{attribute addProperty BoxType "EK1100-0000-0018"}
{attribute addProperty Id "Beckhoff_EL1xxxEK1122Beckhoff_EL1xxxEK1122_BA3F35BD162A_0001_EL1002_0000_0000EL1002_FE5AE676486A_0002_EL1002_0000_0016EL1002_FE5AE676486A_0003_EL1002_0000_0017EL1002_FE5AE676486A_0004_EL1002_0000_0018EL1002_FE5AE676486A_0005_EL1004_0000_0000EL1004_5A15FBDA648A_0006_EL1004_0000_0016EL1004_5A15FBDA648A_0007_EL1004_0000_0017EL1004_5A15FBDA648A_0008_EL1004_0000_0018EL1004_5A15FBDA648A_0009_EL1004_0000_0019EL1004_5A15FBDA648A_0010_EL1004_0010_0000EL1004_5A15FBDA648A_0011_EL1004_0010_0016EL1004_5A15FBDA648A_0012_EL1004_0010_0017EL1004_5A15FBDA648A_0013_EL1004_0010_0018EL1004_5A15FBDA648A_0014_EL1004_0020_0016EL1004_5A15FBDA648A_0015_EL1008_0000_0016EL1008_C6161DDF9612A_0016_EL1008_0000_0017EL1008_C6161DDF9612A_0017_EL1008_0000_0018EL1008_C6161DDF9612A_0018_EL1012_0000_0000EL1012_FE5AE676486A_0019_EL1012_0000_0016EL1012_FE5AE676486A_0020_EL1012_0000_0017EL1012_FE5AE676486A_0021_EL1012_0000_0018EL1012_FE5AE676486A_0022_EL1014_0000_0000EL1014_5A15FBDA648A_0023_EL1014_0000_0016EL1014_5A15FBDA648A_0024_EL1014_0000_0017EL1014_5A15FBDA648A_0025_EL1014_0000_0018EL1014_5A15FBDA648A_0026_EL1014_0000_0019EL1014_5A15FBDA648A_0027_EL1014_0010_0000EL1014_5A15FBDA648A_0028_EL1014_0010_0016EL1014_5A15FBDA648A_0029_EL1014_0010_0017EL1014_5A15FBDA648A_0030_EL1014_0010_0018EL1014_5A15FBDA648A_0031_EL1014_0010_0019EL1014_5A15FBDA648A_0032_EL1018_0000_0016EL1018_C6161DDF9612A_0033_EL1018_0000_0017EL1018_C6161DDF9612A_0034_EL1018_0000_0018EL1018_C6161DDF9612A_0035_EL1024_0000_0016EL1024_5A15FBDA648A_0036_EL1024_0000_0017EL1024_5A15FBDA648A_0037_EL1024_0000_0018EL1024_5A15FBDA648A_0038_EL1034_0000_0016EL1034_5A15FBDA648A_0039_EL1034_0000_0017EL1034_5A15FBDA648A_0040_EL1034_0000_0018EL1034_5A15FBDA648A_0041_EL1052_0000_0016EL1052_0A1DBF07648A_0042_EL1054_0000_0016EL1054_0581C7AF9612A_0043_EL1084_0000_0016EL1084_5A15FBDA648A_0044_EL1084_0000_0017EL1084_5A15FBDA648A_0045_EL1084_0000_0018EL1084_5A15FBDA648A_0046_EL1088_0000_0016EL1088_C6161DDF9612A_0047_EL1088_0000_0017EL1088_C6161DDF9612A_0048_EL1088_0000_0018EL1088_C6161DDF9612A_0049_EL1094_0000_0016EL1094_5A15FBDA648A_0050_EL1094_0000_0017EL1094_5A15FBDA648A_0051_EL1094_0000_0018EL1094_5A15FBDA648A_0052_EL1098_0000_0016EL1098_C6161DDF9612A_0053_EL1098_0000_0017EL1098_C6161DDF9612A_0054_EL1098_0000_0018EL1098_C6161DDF9612A_0055_EL1104_0000_0016EL1104_5A15FBDA648A_0056_EL1104_0000_0017EL1104_5A15FBDA648A_0057_EL1104_0000_0018EL1104_5A15FBDA648A_0058_EL1114_0000_0016EL1114_5A15FBDA648A_0059_EL1114_0000_0017EL1114_5A15FBDA648A_0060_EL1114_0000_0018EL1114_5A15FBDA648A_0061_EL1124_0000_0016EL1124_5A15FBDA648A_0062_EL1124_0000_0017EL1124_5A15FBDA648A_0063_EL1124_0000_0018EL1124_5A15FBDA648A_0064_EL1134_0000_0016EL1134_5A15FBDA648A_0065_EL1134_0000_0017EL1134_5A15FBDA648A_0066_EL1134_0000_0018EL1134_5A15FBDA648A_0067_EL1144_0000_0016EL1144_5A15FBDA648A_0068_EL1144_0000_0017EL1144_5A15FBDA648A_0069_EL1144_0000_0018EL1144_5A15FBDA648A_0070_EL1202_0000_0016EL1202_FE5AE676486A_0071_EL1202_0000_0017EL1202_FE5AE676486A_0072_EL1202_0000_0018EL1202_FE5AE676486A_0073_EL1202_0000_0019EL1202_FE5AE676486A_0074_EL1202_0100_0016EL1202_3E03878817622A_0075_EL1202_0100_0017EL1202_3E03878817622A_0076_EL1202_0100_0018EL1202_3E03878817622A_0077_EL1202_0100_0019EL1202_3E03878817622A_0078_EL1252_0000_0017EL1252_30076DEE38448A_0079_EL1252_0000_0018EL1252_54261E5238448A_0080_EL1252_0000_0019EL1252_54261E5238448A_0081_EL1252_0000_0020EL1252_54261E5238448A_0082_EL1252_0000_0021EL1252_54261E5238448A_0083_EL1252_0000_0022EL1252_54261E5238448A_0084_EL1252_0010_0019EL1252_54261E5238448A_0085_EL1252_0010_0020EL1252_54261E5238448A_0086_EL1252_0010_0021EL1252_54261E5238448A_0087_EL1252_0050_0016EL1252_54261E5238448A_0088_EL1252_0050_0017EL1252_54261E5238448A_0089_EL1252_0050_0018EL1252_54261E5238448A_0090_EL1254_0000_0000EL1254_D71D85A467284A_0091_EL1262_0000_0002EL1262_0572C52632040A_0092_EL1262_0000_0003EL1262_0572C52632040A_0093_EL1262_0050_0002EL1262_0572C52632040A_0094_EL1262_0050_0003EL1262_0572C52632040A_0095_EL1258_0000_0016EL1258_54C5F1D75784723A_0096_EL1258_0000_0017EL1258_D5DBF8D73488436A_0097_EL1258_0010_0017EL1258_F90AE7941184148A_0098_EL1259_0000_0016EL1259_07379E76112401405A_0099_EL1259_0000_0017EL1259_CA442E63111841398A_0100_EL1259_0000_0018EL1259_0CA51D3C101201265A_0101_EL1382_0000_0016EL1382_0A1DBF07648A_0102_EL1382_0000_0017EL1382_0A1DBF07648A_0103_EL1382_0000_0018EL1382_0A1DBF07648A_0104_EL1702_0000_0016EL1702_FE5AE676486A_0105_EL1702_0000_0017EL1702_FE5AE676486A_0106_EL1702_0020_0016EL1702_FE5AE676486A_0107_EL1712_0000_0016EL1712_FE5AE676486A_0108_EL1712_0020_0016EL1712_FE5AE676486A_0109_EL1722_0000_0016EL1722_FE5AE676486A_0110_EL1722_0000_0017EL1722_FE5AE676486A_0111_EL1804_0000_0016EL1804_5A15FBDA648A_0112_EL1804_0000_0017EL1804_5A15FBDA648A_0113_EL1804_0000_0018EL1804_5A15FBDA648A_0114_EL1808_0000_0016EL1808_C6161DDF9612A_0115_EL1808_0000_0017EL1808_C6161DDF9612A_0116_EL1808_0000_0018EL1808_C6161DDF9612A_0117_EL1809_0000_0016EL1809_8059E62316020A_0118_EL1809_0000_0017EL1809_8059E62316020A_0119_EL1809_0000_0018EL1809_8059E62316020A_0120_EL1814_0000_0016EL1814_5A15FBDA648A_0121_EL1814_0000_0017EL1814_5A15FBDA648A_0122_EL1814_0000_0018EL1814_5A15FBDA648A_0123_EL1819_0000_0016EL1819_8059E62316020A_0124_EL1819_0000_0017EL1819_8059E62316020A_0125_EL1819_0000_0018EL1819_8059E62316020A_0126_EL1852_0000_0016EL1852_6598BC3916020A_0127_EL1859_0000_0016EL1859_6598BC3916020A_0128_EL1859_0000_0017EL1859_6598BC3916020A_0129_EL1859_0000_0018EL1859_6598BC3916020A_0130_EL1862_0000_0016EL1862_8059E62316020A_0131_EL1862_0000_0017EL1862_8059E62316020A_0132_EL1862_0000_0018EL1862_8059E62316020A_0133_EL1862_0000_0019EL1862_8059E62316020A_0134_EL1862_0010_0016EL1862_8059E62316020A_0135_EL1862_0010_0017EL1862_8059E62316020A_0136_EL1862_0010_0018EL1862_8059E62316020A_0137_EL1862_0010_0019EL1862_8059E62316020A_0138_EL1872_0000_0016EL1872_8059E62316020A_0139_EL1872_0000_0017EL1872_8059E62316020A_0140_EL1872_0000_0018EL1872_8059E62316020A_0141_EL1872_0010_0016EL1872_8059E62316020A_0142_EL1889_0000_0016EL1889_8059E62316020A_0143_EL1889_0000_0017EL1889_8059E62316020A_0144_EL1889_0000_0018EL1889_8059E62316020A_0145_EL1889_0000_0019EL1889_8059E62316020A_0146_EL1899_0000_0016EL1899_8059E62316020"}
{attribute addProperty CRC "2019569491"}
{attribute addProperty SizeInBites "60696"}
{attribute addProperty SizeInBytes "7587"}
TYPE Beckhoff_EL1xxx_78602F53 EXTENDS EK1100_179A0949 :
STRUCT
	{attribute addProperty Name "Beckhoff_EL1xxxEK1122"}
	Beckhoff_EL1xxxEK1122 : Beckhoff_EL1xxxEK1122_BA3F35BD;
	{attribute addProperty Name "A_0001_EL1002_0000_0000"}
	A_0001_EL1002_0000_0000 : EL1002_FE5AE676;
	{attribute addProperty Name "A_0002_EL1002_0000_0016"}
	A_0002_EL1002_0000_0016 : EL1002_FE5AE676;
	{attribute addProperty Name "A_0003_EL1002_0000_0017"}
	A_0003_EL1002_0000_0017 : EL1002_FE5AE676;
	{attribute addProperty Name "A_0004_EL1002_0000_0018"}
	A_0004_EL1002_0000_0018 : EL1002_FE5AE676;
	{attribute addProperty Name "A_0005_EL1004_0000_0000"}
	A_0005_EL1004_0000_0000 : EL1004_5A15FBDA;
	{attribute addProperty Name "A_0006_EL1004_0000_0016"}
	A_0006_EL1004_0000_0016 : EL1004_5A15FBDA;
	{attribute addProperty Name "A_0007_EL1004_0000_0017"}
	A_0007_EL1004_0000_0017 : EL1004_5A15FBDA;
	{attribute addProperty Name "A_0008_EL1004_0000_0018"}
	A_0008_EL1004_0000_0018 : EL1004_5A15FBDA;
	{attribute addProperty Name "A_0009_EL1004_0000_0019"}
	A_0009_EL1004_0000_0019 : EL1004_5A15FBDA;
	{attribute addProperty Name "A_0010_EL1004_0010_0000"}
	A_0010_EL1004_0010_0000 : EL1004_5A15FBDA;
	{attribute addProperty Name "A_0011_EL1004_0010_0016"}
	A_0011_EL1004_0010_0016 : EL1004_5A15FBDA;
	{attribute addProperty Name "A_0012_EL1004_0010_0017"}
	A_0012_EL1004_0010_0017 : EL1004_5A15FBDA;
	{attribute addProperty Name "A_0013_EL1004_0010_0018"}
	A_0013_EL1004_0010_0018 : EL1004_5A15FBDA;
	{attribute addProperty Name "A_0014_EL1004_0020_0016"}
	A_0014_EL1004_0020_0016 : EL1004_5A15FBDA;
	{attribute addProperty Name "A_0015_EL1008_0000_0016"}
	A_0015_EL1008_0000_0016 : EL1008_C6161DDF;
	{attribute addProperty Name "A_0016_EL1008_0000_0017"}
	A_0016_EL1008_0000_0017 : EL1008_C6161DDF;
	{attribute addProperty Name "A_0017_EL1008_0000_0018"}
	A_0017_EL1008_0000_0018 : EL1008_C6161DDF;
	{attribute addProperty Name "A_0018_EL1012_0000_0000"}
	A_0018_EL1012_0000_0000 : EL1012_FE5AE676;
	{attribute addProperty Name "A_0019_EL1012_0000_0016"}
	A_0019_EL1012_0000_0016 : EL1012_FE5AE676;
	{attribute addProperty Name "A_0020_EL1012_0000_0017"}
	A_0020_EL1012_0000_0017 : EL1012_FE5AE676;
	{attribute addProperty Name "A_0021_EL1012_0000_0018"}
	A_0021_EL1012_0000_0018 : EL1012_FE5AE676;
	{attribute addProperty Name "A_0022_EL1014_0000_0000"}
	A_0022_EL1014_0000_0000 : EL1014_5A15FBDA;
	{attribute addProperty Name "A_0023_EL1014_0000_0016"}
	A_0023_EL1014_0000_0016 : EL1014_5A15FBDA;
	{attribute addProperty Name "A_0024_EL1014_0000_0017"}
	A_0024_EL1014_0000_0017 : EL1014_5A15FBDA;
	{attribute addProperty Name "A_0025_EL1014_0000_0018"}
	A_0025_EL1014_0000_0018 : EL1014_5A15FBDA;
	{attribute addProperty Name "A_0026_EL1014_0000_0019"}
	A_0026_EL1014_0000_0019 : EL1014_5A15FBDA;
	{attribute addProperty Name "A_0027_EL1014_0010_0000"}
	A_0027_EL1014_0010_0000 : EL1014_5A15FBDA;
	{attribute addProperty Name "A_0028_EL1014_0010_0016"}
	A_0028_EL1014_0010_0016 : EL1014_5A15FBDA;
	{attribute addProperty Name "A_0029_EL1014_0010_0017"}
	A_0029_EL1014_0010_0017 : EL1014_5A15FBDA;
	{attribute addProperty Name "A_0030_EL1014_0010_0018"}
	A_0030_EL1014_0010_0018 : EL1014_5A15FBDA;
	{attribute addProperty Name "A_0031_EL1014_0010_0019"}
	A_0031_EL1014_0010_0019 : EL1014_5A15FBDA;
	{attribute addProperty Name "A_0032_EL1018_0000_0016"}
	A_0032_EL1018_0000_0016 : EL1018_C6161DDF;
	{attribute addProperty Name "A_0033_EL1018_0000_0017"}
	A_0033_EL1018_0000_0017 : EL1018_C6161DDF;
	{attribute addProperty Name "A_0034_EL1018_0000_0018"}
	A_0034_EL1018_0000_0018 : EL1018_C6161DDF;
	{attribute addProperty Name "A_0035_EL1024_0000_0016"}
	A_0035_EL1024_0000_0016 : EL1024_5A15FBDA;
	{attribute addProperty Name "A_0036_EL1024_0000_0017"}
	A_0036_EL1024_0000_0017 : EL1024_5A15FBDA;
	{attribute addProperty Name "A_0037_EL1024_0000_0018"}
	A_0037_EL1024_0000_0018 : EL1024_5A15FBDA;
	{attribute addProperty Name "A_0038_EL1034_0000_0016"}
	A_0038_EL1034_0000_0016 : EL1034_5A15FBDA;
	{attribute addProperty Name "A_0039_EL1034_0000_0017"}
	A_0039_EL1034_0000_0017 : EL1034_5A15FBDA;
	{attribute addProperty Name "A_0040_EL1034_0000_0018"}
	A_0040_EL1034_0000_0018 : EL1034_5A15FBDA;
	{attribute addProperty Name "A_0041_EL1052_0000_0016"}
	A_0041_EL1052_0000_0016 : EL1052_0A1DBF07;
	{attribute addProperty Name "A_0042_EL1054_0000_0016"}
	A_0042_EL1054_0000_0016 : EL1054_0581C7AF;
	{attribute addProperty Name "A_0043_EL1084_0000_0016"}
	A_0043_EL1084_0000_0016 : EL1084_5A15FBDA;
	{attribute addProperty Name "A_0044_EL1084_0000_0017"}
	A_0044_EL1084_0000_0017 : EL1084_5A15FBDA;
	{attribute addProperty Name "A_0045_EL1084_0000_0018"}
	A_0045_EL1084_0000_0018 : EL1084_5A15FBDA;
	{attribute addProperty Name "A_0046_EL1088_0000_0016"}
	A_0046_EL1088_0000_0016 : EL1088_C6161DDF;
	{attribute addProperty Name "A_0047_EL1088_0000_0017"}
	A_0047_EL1088_0000_0017 : EL1088_C6161DDF;
	{attribute addProperty Name "A_0048_EL1088_0000_0018"}
	A_0048_EL1088_0000_0018 : EL1088_C6161DDF;
	{attribute addProperty Name "A_0049_EL1094_0000_0016"}
	A_0049_EL1094_0000_0016 : EL1094_5A15FBDA;
	{attribute addProperty Name "A_0050_EL1094_0000_0017"}
	A_0050_EL1094_0000_0017 : EL1094_5A15FBDA;
	{attribute addProperty Name "A_0051_EL1094_0000_0018"}
	A_0051_EL1094_0000_0018 : EL1094_5A15FBDA;
	{attribute addProperty Name "A_0052_EL1098_0000_0016"}
	A_0052_EL1098_0000_0016 : EL1098_C6161DDF;
	{attribute addProperty Name "A_0053_EL1098_0000_0017"}
	A_0053_EL1098_0000_0017 : EL1098_C6161DDF;
	{attribute addProperty Name "A_0054_EL1098_0000_0018"}
	A_0054_EL1098_0000_0018 : EL1098_C6161DDF;
	{attribute addProperty Name "A_0055_EL1104_0000_0016"}
	A_0055_EL1104_0000_0016 : EL1104_5A15FBDA;
	{attribute addProperty Name "A_0056_EL1104_0000_0017"}
	A_0056_EL1104_0000_0017 : EL1104_5A15FBDA;
	{attribute addProperty Name "A_0057_EL1104_0000_0018"}
	A_0057_EL1104_0000_0018 : EL1104_5A15FBDA;
	{attribute addProperty Name "A_0058_EL1114_0000_0016"}
	A_0058_EL1114_0000_0016 : EL1114_5A15FBDA;
	{attribute addProperty Name "A_0059_EL1114_0000_0017"}
	A_0059_EL1114_0000_0017 : EL1114_5A15FBDA;
	{attribute addProperty Name "A_0060_EL1114_0000_0018"}
	A_0060_EL1114_0000_0018 : EL1114_5A15FBDA;
	{attribute addProperty Name "A_0061_EL1124_0000_0016"}
	A_0061_EL1124_0000_0016 : EL1124_5A15FBDA;
	{attribute addProperty Name "A_0062_EL1124_0000_0017"}
	A_0062_EL1124_0000_0017 : EL1124_5A15FBDA;
	{attribute addProperty Name "A_0063_EL1124_0000_0018"}
	A_0063_EL1124_0000_0018 : EL1124_5A15FBDA;
	{attribute addProperty Name "A_0064_EL1134_0000_0016"}
	A_0064_EL1134_0000_0016 : EL1134_5A15FBDA;
	{attribute addProperty Name "A_0065_EL1134_0000_0017"}
	A_0065_EL1134_0000_0017 : EL1134_5A15FBDA;
	{attribute addProperty Name "A_0066_EL1134_0000_0018"}
	A_0066_EL1134_0000_0018 : EL1134_5A15FBDA;
	{attribute addProperty Name "A_0067_EL1144_0000_0016"}
	A_0067_EL1144_0000_0016 : EL1144_5A15FBDA;
	{attribute addProperty Name "A_0068_EL1144_0000_0017"}
	A_0068_EL1144_0000_0017 : EL1144_5A15FBDA;
	{attribute addProperty Name "A_0069_EL1144_0000_0018"}
	A_0069_EL1144_0000_0018 : EL1144_5A15FBDA;
	{attribute addProperty Name "A_0070_EL1202_0000_0016"}
	A_0070_EL1202_0000_0016 : EL1202_FE5AE676;
	{attribute addProperty Name "A_0071_EL1202_0000_0017"}
	A_0071_EL1202_0000_0017 : EL1202_FE5AE676;
	{attribute addProperty Name "A_0072_EL1202_0000_0018"}
	A_0072_EL1202_0000_0018 : EL1202_FE5AE676;
	{attribute addProperty Name "A_0073_EL1202_0000_0019"}
	A_0073_EL1202_0000_0019 : EL1202_FE5AE676;
	{attribute addProperty Name "A_0074_EL1202_0100_0016"}
	A_0074_EL1202_0100_0016 : EL1202_3E038788;
	{attribute addProperty Name "A_0075_EL1202_0100_0017"}
	A_0075_EL1202_0100_0017 : EL1202_3E038788;
	{attribute addProperty Name "A_0076_EL1202_0100_0018"}
	A_0076_EL1202_0100_0018 : EL1202_3E038788;
	{attribute addProperty Name "A_0077_EL1202_0100_0019"}
	A_0077_EL1202_0100_0019 : EL1202_3E038788;
	{attribute addProperty Name "A_0078_EL1252_0000_0017"}
	A_0078_EL1252_0000_0017 : EL1252_30076DEE;
	{attribute addProperty Name "A_0079_EL1252_0000_0018"}
	A_0079_EL1252_0000_0018 : EL1252_54261E52;
	{attribute addProperty Name "A_0080_EL1252_0000_0019"}
	A_0080_EL1252_0000_0019 : EL1252_54261E52;
	{attribute addProperty Name "A_0081_EL1252_0000_0020"}
	A_0081_EL1252_0000_0020 : EL1252_54261E52;
	{attribute addProperty Name "A_0082_EL1252_0000_0021"}
	A_0082_EL1252_0000_0021 : EL1252_54261E52;
	{attribute addProperty Name "A_0083_EL1252_0000_0022"}
	A_0083_EL1252_0000_0022 : EL1252_54261E52;
	{attribute addProperty Name "A_0084_EL1252_0010_0019"}
	A_0084_EL1252_0010_0019 : EL1252_54261E52;
	{attribute addProperty Name "A_0085_EL1252_0010_0020"}
	A_0085_EL1252_0010_0020 : EL1252_54261E52;
	{attribute addProperty Name "A_0086_EL1252_0010_0021"}
	A_0086_EL1252_0010_0021 : EL1252_54261E52;
	{attribute addProperty Name "A_0087_EL1252_0050_0016"}
	A_0087_EL1252_0050_0016 : EL1252_54261E52;
	{attribute addProperty Name "A_0088_EL1252_0050_0017"}
	A_0088_EL1252_0050_0017 : EL1252_54261E52;
	{attribute addProperty Name "A_0089_EL1252_0050_0018"}
	A_0089_EL1252_0050_0018 : EL1252_54261E52;
	{attribute addProperty Name "A_0090_EL1254_0000_0000"}
	A_0090_EL1254_0000_0000 : EL1254_D71D85A4;
	{attribute addProperty Name "A_0091_EL1262_0000_0002"}
	A_0091_EL1262_0000_0002 : EL1262_0572C526;
	{attribute addProperty Name "A_0092_EL1262_0000_0003"}
	A_0092_EL1262_0000_0003 : EL1262_0572C526;
	{attribute addProperty Name "A_0093_EL1262_0050_0002"}
	A_0093_EL1262_0050_0002 : EL1262_0572C526;
	{attribute addProperty Name "A_0094_EL1262_0050_0003"}
	A_0094_EL1262_0050_0003 : EL1262_0572C526;
	{attribute addProperty Name "A_0095_EL1258_0000_0016"}
	A_0095_EL1258_0000_0016 : EL1258_54C5F1D7;
	{attribute addProperty Name "A_0096_EL1258_0000_0017"}
	A_0096_EL1258_0000_0017 : EL1258_D5DBF8D7;
	{attribute addProperty Name "A_0097_EL1258_0010_0017"}
	A_0097_EL1258_0010_0017 : EL1258_F90AE794;
	{attribute addProperty Name "A_0098_EL1259_0000_0016"}
	A_0098_EL1259_0000_0016 : EL1259_07379E76;
	{attribute addProperty Name "A_0099_EL1259_0000_0017"}
	A_0099_EL1259_0000_0017 : EL1259_CA442E63;
	{attribute addProperty Name "A_0100_EL1259_0000_0018"}
	A_0100_EL1259_0000_0018 : EL1259_0CA51D3C;
	{attribute addProperty Name "A_0101_EL1382_0000_0016"}
	A_0101_EL1382_0000_0016 : EL1382_0A1DBF07;
	{attribute addProperty Name "A_0102_EL1382_0000_0017"}
	A_0102_EL1382_0000_0017 : EL1382_0A1DBF07;
	{attribute addProperty Name "A_0103_EL1382_0000_0018"}
	A_0103_EL1382_0000_0018 : EL1382_0A1DBF07;
	{attribute addProperty Name "A_0104_EL1702_0000_0016"}
	A_0104_EL1702_0000_0016 : EL1702_FE5AE676;
	{attribute addProperty Name "A_0105_EL1702_0000_0017"}
	A_0105_EL1702_0000_0017 : EL1702_FE5AE676;
	{attribute addProperty Name "A_0106_EL1702_0020_0016"}
	A_0106_EL1702_0020_0016 : EL1702_FE5AE676;
	{attribute addProperty Name "A_0107_EL1712_0000_0016"}
	A_0107_EL1712_0000_0016 : EL1712_FE5AE676;
	{attribute addProperty Name "A_0108_EL1712_0020_0016"}
	A_0108_EL1712_0020_0016 : EL1712_FE5AE676;
	{attribute addProperty Name "A_0109_EL1722_0000_0016"}
	A_0109_EL1722_0000_0016 : EL1722_FE5AE676;
	{attribute addProperty Name "A_0110_EL1722_0000_0017"}
	A_0110_EL1722_0000_0017 : EL1722_FE5AE676;
	{attribute addProperty Name "A_0111_EL1804_0000_0016"}
	A_0111_EL1804_0000_0016 : EL1804_5A15FBDA;
	{attribute addProperty Name "A_0112_EL1804_0000_0017"}
	A_0112_EL1804_0000_0017 : EL1804_5A15FBDA;
	{attribute addProperty Name "A_0113_EL1804_0000_0018"}
	A_0113_EL1804_0000_0018 : EL1804_5A15FBDA;
	{attribute addProperty Name "A_0114_EL1808_0000_0016"}
	A_0114_EL1808_0000_0016 : EL1808_C6161DDF;
	{attribute addProperty Name "A_0115_EL1808_0000_0017"}
	A_0115_EL1808_0000_0017 : EL1808_C6161DDF;
	{attribute addProperty Name "A_0116_EL1808_0000_0018"}
	A_0116_EL1808_0000_0018 : EL1808_C6161DDF;
	{attribute addProperty Name "A_0117_EL1809_0000_0016"}
	A_0117_EL1809_0000_0016 : EL1809_8059E623;
	{attribute addProperty Name "A_0118_EL1809_0000_0017"}
	A_0118_EL1809_0000_0017 : EL1809_8059E623;
	{attribute addProperty Name "A_0119_EL1809_0000_0018"}
	A_0119_EL1809_0000_0018 : EL1809_8059E623;
	{attribute addProperty Name "A_0120_EL1814_0000_0016"}
	A_0120_EL1814_0000_0016 : EL1814_5A15FBDA;
	{attribute addProperty Name "A_0121_EL1814_0000_0017"}
	A_0121_EL1814_0000_0017 : EL1814_5A15FBDA;
	{attribute addProperty Name "A_0122_EL1814_0000_0018"}
	A_0122_EL1814_0000_0018 : EL1814_5A15FBDA;
	{attribute addProperty Name "A_0123_EL1819_0000_0016"}
	A_0123_EL1819_0000_0016 : EL1819_8059E623;
	{attribute addProperty Name "A_0124_EL1819_0000_0017"}
	A_0124_EL1819_0000_0017 : EL1819_8059E623;
	{attribute addProperty Name "A_0125_EL1819_0000_0018"}
	A_0125_EL1819_0000_0018 : EL1819_8059E623;
	{attribute addProperty Name "A_0126_EL1852_0000_0016"}
	A_0126_EL1852_0000_0016 : EL1852_6598BC39;
	{attribute addProperty Name "A_0127_EL1859_0000_0016"}
	A_0127_EL1859_0000_0016 : EL1859_6598BC39;
	{attribute addProperty Name "A_0128_EL1859_0000_0017"}
	A_0128_EL1859_0000_0017 : EL1859_6598BC39;
	{attribute addProperty Name "A_0129_EL1859_0000_0018"}
	A_0129_EL1859_0000_0018 : EL1859_6598BC39;
	{attribute addProperty Name "A_0130_EL1862_0000_0016"}
	A_0130_EL1862_0000_0016 : EL1862_8059E623;
	{attribute addProperty Name "A_0131_EL1862_0000_0017"}
	A_0131_EL1862_0000_0017 : EL1862_8059E623;
	{attribute addProperty Name "A_0132_EL1862_0000_0018"}
	A_0132_EL1862_0000_0018 : EL1862_8059E623;
	{attribute addProperty Name "A_0133_EL1862_0000_0019"}
	A_0133_EL1862_0000_0019 : EL1862_8059E623;
	{attribute addProperty Name "A_0134_EL1862_0010_0016"}
	A_0134_EL1862_0010_0016 : EL1862_8059E623;
	{attribute addProperty Name "A_0135_EL1862_0010_0017"}
	A_0135_EL1862_0010_0017 : EL1862_8059E623;
	{attribute addProperty Name "A_0136_EL1862_0010_0018"}
	A_0136_EL1862_0010_0018 : EL1862_8059E623;
	{attribute addProperty Name "A_0137_EL1862_0010_0019"}
	A_0137_EL1862_0010_0019 : EL1862_8059E623;
	{attribute addProperty Name "A_0138_EL1872_0000_0016"}
	A_0138_EL1872_0000_0016 : EL1872_8059E623;
	{attribute addProperty Name "A_0139_EL1872_0000_0017"}
	A_0139_EL1872_0000_0017 : EL1872_8059E623;
	{attribute addProperty Name "A_0140_EL1872_0000_0018"}
	A_0140_EL1872_0000_0018 : EL1872_8059E623;
	{attribute addProperty Name "A_0141_EL1872_0010_0016"}
	A_0141_EL1872_0010_0016 : EL1872_8059E623;
	{attribute addProperty Name "A_0142_EL1889_0000_0016"}
	A_0142_EL1889_0000_0016 : EL1889_8059E623;
	{attribute addProperty Name "A_0143_EL1889_0000_0017"}
	A_0143_EL1889_0000_0017 : EL1889_8059E623;
	{attribute addProperty Name "A_0144_EL1889_0000_0018"}
	A_0144_EL1889_0000_0018 : EL1889_8059E623;
	{attribute addProperty Name "A_0145_EL1889_0000_0019"}
	A_0145_EL1889_0000_0019 : EL1889_8059E623;
	{attribute addProperty Name "A_0146_EL1899_0000_0016"}
	A_0146_EL1899_0000_0016 : EL1899_8059E623;
END_STRUCT
END_TYPE

(* stored: Version 1.2.0.0, ProductVersion 3.1.4024.9
   DUT Beckhoff_EL1xxx_78602F53: Id {403ae7cd-692d-4301-8fab-d61561667fb2} *)
